// TIA Portal V20 export
VAR_GLOBAL   // PLC tag table "LGR_Const_LogClass"
END_VAR
VAR_GLOBAL CONSTANT   // user constants
   "LEVEL.DEBUG" : UInt := 1;
   "LEVEL.INFO" : UInt := 5;
   "LEVEL.WARN" : UInt := 7;
   "LEVEL.ERROR" : UInt := 8;
   "LEVEL.FATAL" : UInt := 9;
   "SOURCE.SAFETY" : UInt := 90;
   "SOURCE.PLC" : UInt := 80;
   "SOURCE.DRIVE" : UInt := 70;
   "SOURCE.PARA" : UInt := 60;
   "SOURCE.LOGIC" : UInt := 50;
   "SOURCE.INTERFACE" : UInt := 40;
   "SOURCE.COMMUNICATION" : UInt := 30;
   "SOURCE.GCS" : UInt := 20;
   "SOURCE.COMMON" : UInt := 10;
   "COMMAND.INIT" : UInt := 1;
   "COMMAND.JOG" : UInt := 10;
   "COMMAND.POWERON" : UInt := 3;
   "COMMAND.DRIVEON" : UInt := 4;
   "COMMAND.SETORIGIN" : UInt := 5;
   "COMMAND.PROC" : UInt := 30;
   "COMMAND.GCS" : UInt := 50;
   "COMMAND.MODE" : UInt := 2;
   "PROC.LOG.START" : UInt := 1;
   "PROC.LOG.DONE" : UInt := 2;
   "PROC.LOG.STOP" : UInt := 3;
   "PROC.LOG.RESUME" : UInt := 4;
   "GCS.CMD.EXECUTED" : UInt := 1;
   "GCS.CMD.REJECTED" : UInt := 2;
   "GCS.CMD.UNDEFINED" : UInt := 3;
   "COMMAND.FAULT" : UInt := 90;
   "PROC.LOG.GCSRECV" : UInt := 5;
   "SOURCE.SENSOR" : UInt := 51;
   "SOURCE.COMPONENT" : UInt := 91;
   "COMMAND.TASK" : UInt := 32;
   "COMMAND.STEP" : UInt := 31;
   "COMMAND.WARN" : UInt := 91;
END_VAR
